{attribute 'GeneratedUsingTerminal: EJ2502-0000-0023'}
{attribute addProperty BoxType "EJ2502-0000-0023"}
{attribute addProperty Id "PWM_Outputs_Channel_1AT %Q*PWM_Outputs_Channel_4C6289CD2PWM_Outputs_Channel_2AT %Q*PWM_Outputs_Channel_4C6289CD2WcStateAT %I*WcState_0B2B16F91InfoDataAT %I*InfoData_32EB74EA10"}
{attribute addProperty CRC "4263597303"}
{attribute addProperty Size "15"}
TYPE EJ2502_FE2154F7 :
STRUCT
	{attribute addProperty Name "PWM_Outputs_Channel_1"}
	PWM_Outputs_Channel_1 : PWM_Outputs_Channel_4C6289CD;
	{attribute addProperty Name "PWM_Outputs_Channel_2"}
	PWM_Outputs_Channel_2 : PWM_Outputs_Channel_4C6289CD;
	{attribute addProperty Name "WcState"}
	WcState : WcState_0B2B16F9;
	{attribute addProperty Name "InfoData"}
	InfoData : InfoData_32EB74EA;
END_STRUCT
END_TYPE

(* stored: Version 1.2.0.0, ProductVersion 3.1.4024.9
   DUT EJ2502_FE2154F7: Id {b7c4fb68-0f7b-411a-ab24-9ca028d3d552} *)
